// TIA Portal V20 export
FUNCTION_BLOCK "FB_Consecutive"   // FB90, SCL
{ S7_Optimized_Access := 'TRUE' }
// stored: MemoryReserve 100, SetENOAutomatically false
   VAR_INPUT
      iReset : Bool;
      iGoodEntry : Bool;
      iBadEntry : Bool;
      iPresetValue : Int;
   END_VAR
   VAR_OUTPUT
      oConsecutiveError : Bool;
   END_VAR
   VAR
      sConsecutiveCounter : Int;
      sRT_GoodEntry : R_TRIG;
      sRT_BadEntry { S7_SetPoint := 'True'} : R_TRIG;
   END_VAR
BEGIN
   REGION Description header 
       //==================================================================================
       // POSALUX Swiss SA / (C) Copyright 2026
       //----------------------------------------------------------------------------------
       // Title: FB_Consecutive
       // Comment/Function: 
       // Author: Fabien WALDT
       // Engineering: TIA Portal v20
       //----------------------------------------------------------------------------------
       // Change log table:
       // Version  | Date     | Expert in charge | Changes applied
       // ---------|----------|------------------|-----------------------------------------
       // 00.00.01 | 20260401 | WFA              | First released version
       // =================================================================================
   END_REGION

   REGION R_Trig
       #sRT_GoodEntry(CLK := #iGoodEntry);
       #sRT_BadEntry(CLK := #iBadEntry);
   END_REGION

   REGION Consecutive Counter
       IF #sRT_GoodEntry.Q OR #iReset THEN
           #oConsecutiveError := FALSE;
           #sConsecutiveCounter := 0;
       END_IF;

       IF #sRT_BadEntry.Q THEN
           #sConsecutiveCounter := #sConsecutiveCounter + 1;
       END_IF;

       IF #sConsecutiveCounter >= #iPresetValue THEN
           #oConsecutiveError := TRUE;
       END_IF;
   END_REGION
END_FUNCTION_BLOCK
